SUBAPPLICATION GreenWhiteBackground_Licht (* Subapplication Type *)
  (* Standard: 61499-2 *)
  (* Version 1.0, 2023-02-11, franz *)
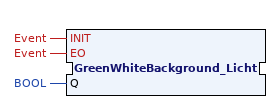
  EVENT_INPUT
    INIT;
    EO;
  END_EVENT
  VAR_INPUT
    Q : BOOL;
  END_VAR
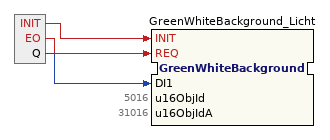
  FBS
    GreenWhiteBackground_Licht : GreenWhiteBackground(u16ObjId := 5016, u16ObjIdA := 31016);
  END_FBS
  EVENT_CONNECTIONS
    INIT TO GreenWhiteBackground_Licht.INIT;
    EO TO GreenWhiteBackground_Licht.REQ;
  END_CONNECTIONS
  DATA_CONNECTIONS
    Q TO GreenWhiteBackground_Licht.DI1;
  END_CONNECTIONS
END_SUBAPPLICATION
